(*
SPDX-FileCopyrightText: © 2026 Oleksandr Tiutyk <trofimich@gmail.com>
SPDX-License-Identifier: MIT
License: https://opensource.org/license/mit
*)

INTERFACE IInvalidNestedWorkflowStateException EXTENDS TOF_Core.IGeneralException

METHOD Throw
VAR_INPUT
	sourceNamespaceName : STRING;
	sourceClassName : STRING;
	sourcePOUName : STRING;
	sourcePosition : STRING;
	nestedActivityState : WORKFLOW_ELEMENT_STATE;
END_VAR
END_METHOD

END_INTERFACE

(* stored: Version 1.1.0.1
   Itf IInvalidNestedWorkflowStateException: Id {795058f3-1af6-4b6d-a614-ac81afb8e1c0}
   Method Throw: Id {1df65ba3-ad31-4a90-9415-a4bd53aaa136} *)
